tmpDataSend[66] := WORD_TO_BYTE(SHR(下卷扬伺服电流, 8));
tmpDataSend[67] := WORD_TO_BYTE(下卷扬伺服电流 AND 16#FF);
tmpDataSend[68] := WORD_TO_BYTE(SHR(下卷扬伺服速度, 8));
tmpDataSend[69] := WORD_TO_BYTE(下卷扬伺服速度 AND 16#FF);
tmpDataSend[70] := WORD_TO_BYTE(SHR(下卷扬伺服位置, 8));
tmpDataSend[71] := WORD_TO_BYTE(下卷扬伺服位置 AND 16#FF);
tmpDataSend[72] := WORD_TO_BYTE(SHR(下卷扬伺服温度, 8));
tmpDataSend[73] := WORD_TO_BYTE(下卷扬伺服温度 AND 16#FF);
tmpDataSend[74] := WORD_TO_BYTE(SHR(下卷扬伺服报错码, 8));
tmpDataSend[75] := WORD_TO_BYTE(下卷扬伺服报错码 AND 16#FF);
tmpDataSend[76] := 16#01;	//0-离线 1-在线

tmpDataSend[77] := WORD_TO_BYTE(SHR(滚刷伺服电流, 8));
tmpDataSend[78] := WORD_TO_BYTE(滚刷伺服电流 AND 16#FF);
tmpDataSend[79] := WORD_TO_BYTE(SHR(滚刷伺服速度, 8));
tmpDataSend[80] := WORD_TO_BYTE(滚刷伺服速度 AND 16#FF);
tmpDataSend[81] := WORD_TO_BYTE(SHR(滚刷伺服温度, 8));
tmpDataSend[82] := WORD_TO_BYTE(滚刷伺服温度 AND 16#FF);
tmpDataSend[83] := WORD_TO_BYTE(SHR(滚刷伺服报错码, 8));
tmpDataSend[84] := WORD_TO_BYTE(滚刷伺服报错码 AND 16#FF);
tmpDataSend[85] := 16#01;	//0-离线 1-在线

tmpDataSend[86] := 16#00;	//风机1启动状态 0-停止 1-启动
tmpDataSend[87] := 16#00;	//风机2启动状态 0-停止 1-启动

tmpDataSend[88] := WORD_TO_BYTE(SHR(左前测距超声波数据, 8));
tmpDataSend[89] := WORD_TO_BYTE(左前测距超声波数据 AND 16#FF);
tmpDataSend[90] := WORD_TO_BYTE(SHR(右前测距超声波数据, 8));
tmpDataSend[97] := WORD_TO_BYTE(右前测距超声波数据 AND 16#FF);
tmpDataSend[92] := WORD_TO_BYTE(SHR(左后测距超声波数据, 8));
tmpDataSend[93] := WORD_TO_BYTE(左后测距超声波数据 AND 16#FF);
tmpDataSend[94] := WORD_TO_BYTE(SHR(右后测距超声波数据, 8));
tmpDataSend[95] := WORD_TO_BYTE(右后测距超声波数据 AND 16#FF);

tmpDataSend[96] := WORD_TO_BYTE(SHR(左前边沿超声波数据, 8));
tmpDataSend[97] := WORD_TO_BYTE(左前边沿超声波数据 AND 16#FF);
tmpDataSend[98] := WORD_TO_BYTE(SHR(右前边沿超声波数据, 8));
tmpDataSend[99] := WORD_TO_BYTE(右前边沿超声波数据 AND 16#FF);
tmpDataSend[100] := WORD_TO_BYTE(SHR(左后边沿超声波数据, 8));
tmpDataSend[101] := WORD_TO_BYTE(左后边沿超声波数据 AND 16#FF);
tmpDataSend[102] := WORD_TO_BYTE(SHR(右后边沿超声波数据, 8));
tmpDataSend[103] := WORD_TO_BYTE(右后边沿超声波数据 AND 16#FF);

tmpDataSend[104] := WORD_TO_BYTE(SHR(机械臂空间X, 8));
tmpDataSend[105] := WORD_TO_BYTE(机械臂空间X AND 16#FF);
tmpDataSend[106] := WORD_TO_BYTE(SHR(机械臂空间Y, 8));
tmpDataSend[107] := WORD_TO_BYTE(机械臂空间Y AND 16#FF);
tmpDataSend[108] := WORD_TO_BYTE(SHR(机械臂空间Z, 8));
tmpDataSend[109] := WORD_TO_BYTE(机械臂空间Z AND 16#FF);
tmpDataSend[110] := WORD_TO_BYTE(SHR(机械臂空间B, 8));
tmpDataSend[111] := WORD_TO_BYTE(机械臂空间B AND 16#FF);
tmpDataSend[112] := WORD_TO_BYTE(SHR(底盘俯仰角, 8));
tmpDataSend[113] := WORD_TO_BYTE(底盘俯仰角 AND 16#FF);
tmpDataSend[114] := WORD_TO_BYTE(SHR(底盘横滚角, 8));
tmpDataSend[115] := WORD_TO_BYTE(底盘横滚角 AND 16#FF);

tmpDataSend[116] := WORD_TO_BYTE(机械臂运行状态); //0-上使能，1-掉使能，2-运行中，3-报错
tmpDataSend[117] := WORD_TO_BYTE(机械臂报错码);

上传信息处理_1(定时时间:=T#0MS, 数据域长度:=118, pInputData:=ADR(tmpDataSend[0]), 应答:=16#00, 序列号:=上传序列号, 主功能码:=16#02, 次功能码:=16#06);
END_METHOD

END_PROGRAM

// Device/Application/函数/运动控制/清扫作业流程
FUNCTION_BLOCK 清扫作业流程
VAR_IN_OUT
	作业状态		: INT;	//0-系统初始化, 10-清扫待命状态, 20-清扫准备状态, 30-清扫暂停状态, 40-行走复位状态, 50-急停状态, 60-进入现场操作模式, 70-退出现场操作模式
END_VAR
VAR_INPUT
	离地高度		: LREAL;
	光伏板角度		: LREAL;
	离车间距		: LREAL;
	清扫方向		: LREAL; //0-左侧, 1-右侧	
END_VAR
VAR_OUTPUT
	返回功能码		: BYTE;
	返回状态		: BYTE;		//0x00-运行中, 0x05-完成, 0x0A-异常
END_VAR
VAR
	机械臂清扫准备状态完成		: BOOL := FALSE;
END_VAR

CASE 作业状态 OF
	0 : //系统初始化
		滚刷伺服参数.运行模式 := 0;
		启动回零自动运行:=FALSE;
		启动对中机构自动运行:=FALSE;
		启动上下扬自动运行:=FALSE;
		作业状态 := 5;
	5:
	    启动回零自动运行:=TRUE;
		作业状态 := 6;
	6:
	    IF 回零工作完成 THEN
			返回功能码 := 16#01;
			返回状态 := 16#05;
	    END_IF
	10 : //清扫待命状态
		启动回零自动运行:=TRUE;
		IF 回零工作完成 THEN
            作业状态 := 11;
	    END_IF
	11 :
		机械臂运行参数.倍率 := 70.0;
		机械臂运行参数.规划模式 := 4;
		机械臂运行参数.是否关节运动 := TRUE;
		IF 清扫方向=1 THEN
			机械臂运行参数.运行点位[0] := 90.0;
		ELSE
			机械臂运行参数.运行点位[0] := -90.0;
		END_IF
		机械臂运行参数.运行点位[1] := -90.0; 机械臂运行参数.运行点位[2] := 180.0;
		机械臂运行参数.运行点位[3] := 50.0; 机械臂运行参数.运行点位[4] := 0.0; 机械臂运行参数.运行点位[5] := 0.0;
		IF sMotionOutputs.iRobStatus = 1 THEN
			机械臂运行启动 := TRUE;
		END_IF
		IF sMotionOutputs.iRobStatus = 3 THEN //运动完成
			返回功能码 := 16#02;
			返回状态 := 16#05;
		END_IF
	20 : //清扫准备状态
		机械臂运行参数.规划模式 := 4;
		机械臂运行参数.是否关节运动 := FALSE;
		IF 清扫方向=1 THEN
			机械臂运行参数.运行点位[1] := 2220.0;
		ELSE
			机械臂运行参数.运行点位[1] := -2220.0;
		END_IF
		机械臂运行参数.运行点位[0] := 0.0; 机械臂运行参数.运行点位[2] := 2000.0;
		机械臂运行参数.运行点位[3] := 40.0; 机械臂运行参数.运行点位[4] := 0.0; 机械臂运行参数.运行点位[5] := 0.0;
		滚刷伺服参数.运行模式 := 0;
		IF sMotionOutputs.iRobStatus = 1 THEN //机械臂运行至光伏板上方
			机械臂运行启动 := TRUE;
		END_IF
		IF sMotionOutputs.iRobStatus = 3 THEN //运动完成
			启动对中机构自动运行:=TRUE;
			作业状态 := 27;
		END_IF
	27:
	    IF 对中工作完成 THEN
			启动上下扬自动运行:=TRUE;
	    	作业状态 := 28;
	    END_IF
	28:
	    IF 上下卷扬工作完成 THEN
	    	作业状态 := 29;
	    END_IF
	29:	//清扫准备状态结束
// 	    滚刷伺服参数.运行方向:=TRUE;
		滚刷伺服参数.运行模式 := 1;
		IF 清扫方向=1 THEN
			滚刷伺服参数.运行方向:=FALSE;
		ELSE
			滚刷伺服参数.运行方向:=TRUE;
		END_IF
		返回功能码 := 16#03;
		返回状态 := 16#05;
	30 : //清扫暂停状态
		滚刷伺服参数.运行模式 := 0;
		//伸缩轴伺服参数.运行模式:=0;
		启动对中机构自动运行:=FALSE;
		启动上下扬自动运行:=FALSE;
		启动回零自动运行:=TRUE;
		IF 回零工作完成 THEN
			返回功能码 := 16#04;
			返回状态 := 16#05;
	    END_IF
	40 : //行走复位状态
		启动回零自动运行:=TRUE;
		IF 回零工作完成 THEN
            作业状态 := 41;
	    END_IF
	41 :
		机械臂运行参数.规划模式 := 4;
		机械臂运行参数.是否关节运动 := TRUE;
		机械臂运行参数.运行点位[0] := 0.0; 机械臂运行参数.运行点位[1] := -90.0; 机械臂运行参数.运行点位[2] := 180.0;
		机械臂运行参数.运行点位[3] := 45.0; 机械臂运行参数.运行点位[4] := 0.0; 机械臂运行参数.运行点位[5] := 0.0;
		IF sMotionOutputs.iRobStatus = 1 THEN
			机械臂运行启动 := TRUE;
		END_IF
		IF sMotionOutputs.iRobStatus = 3 THEN //运动完成
			返回功能码 := 16#05;
			返回状态 := 16#05;
		END_IF
	50 : //急停状态
		左上轮伺服参数.运行模式 := 0; 左下轮伺服参数.运行模式 := 0;
		右上轮伺服参数.运行模式 := 0; 右下轮伺服参数.运行模式 := 0;
	
	100: //无操作
// 		启动对中机构自动运行:=FALSE;
// 		启动上下扬自动运行:=FALSE;
		返回功能码 := 16#00;
		返回状态 := 16#00;
	200: //运行异常
		返回状态 := 16#0A;
ELSE
   滚刷伺服参数.运行模式 :=0;
   启动对中机构自动运行:=FALSE;
   启动上下扬自动运行:=FALSE;
END_CASE

END_FUNCTION_BLOCK

// Device/Application/底盘算法处理
PROGRAM 底盘算法处理
VAR
	iCounter			: INT := 0;
	底盘使能				: BOOL := FALSE;
	底盘联动				: BOOL := TRUE;
	
	底盘平衡处理			: 底盘平衡算法;
	
	左上气缸伺服控制    	: 伺服控制;
	左下气缸伺服控制    	: 伺服控制;
	右上气缸伺服控制    	: 伺服控制;
	右下气缸伺服控制    	: 伺服控制;
	
	左上轮伺服控制    	: 伺服控制;
	左下轮伺服控制    	: 伺服控制;
	右上轮伺服控制    	: 伺服控制;
	右下轮伺服控制    	: 伺服控制;  
END_VAR

底盘陀螺仪.X := DINT_TO_REAL(DWORD_TO_DINT( SHL(WORD_TO_DWORD(底盘陀螺仪.orign_arry[1]), 16) OR WORD_TO_DWORD(底盘陀螺仪.orign_arry[0]) )) / 1000;
底盘陀螺仪.Y := DINT_TO_REAL(DWORD_TO_DINT( SHL(WORD_TO_DWORD(底盘陀螺仪.orign_arry[3]), 16) OR WORD_TO_DWORD(底盘陀螺仪.orign_arry[2]) )) / 1000;
底盘陀螺仪.Z := DINT_TO_REAL(DWORD_TO_DINT( SHL(WORD_TO_DWORD(底盘陀螺仪.orign_arry[5]), 16) OR WORD_TO_DWORD(底盘陀螺仪.orign_arry[4]) )) / 1000;

底盘陀螺仪.角速度X := WORD_TO_REAL(底盘陀螺仪.orign_arry_speed[1]) / 32768 * 2000;
底盘陀螺仪.角速度Y := WORD_TO_REAL(底盘陀螺仪.orign_arry_speed[2]) / 32768 * 2000;
底盘陀螺仪.角速度Z := WORD_TO_REAL(底盘陀螺仪.orign_arry_speed[3]) / 32768 * 2000;

IF 底盘算法运行 THEN
	底盘平衡处理(
		陀螺仪roll:= 底盘陀螺仪.X, 
		陀螺仪pitch:= 底盘陀螺仪.Y, 
		陀螺仪roll速度:= 底盘陀螺仪.角速度X, 
		陀螺仪pitch速度:= 底盘陀螺仪.角速度Y, 
		前左轮实际长度:= 底盘控制.平均数据1,//左上气缸伺服参数.反馈位置, 
		后左轮实际长度:= 底盘控制.平均数据2,//左下气缸伺服参数.反馈位置, 	
		前右轮实际长度:= 底盘控制.平均数据3,//右上气缸伺服参数.反馈位置, 
		后右轮实际长度:= 底盘控制.平均数据4,//右下气缸伺服参数.反馈位置, 
		前左轮行驶速度:= 左上轮伺服参数.指令速度, 
		后左轮行驶速度:= 左下轮伺服参数.指令速度, 	
		前右轮行驶速度:= 右上轮伺服参数.指令速度, 
		后右轮行驶速度:= 右下轮伺服参数.指令速度, 	
		前左轮力:= 左上气缸伺服参数.反馈力矩, 
		后左轮力:= 左下气缸伺服参数.反馈力矩, 
		前右轮力:= 右上气缸伺服参数.反馈力矩, 
		后右轮力:= 右下气缸伺服参数.反馈力矩, 	
		前左轮输出=> 左上气缸伺服参数.运行位置, 
		后左轮输出=> 左下气缸伺服参数.运行位置, 
		前右轮输出=> 右上气缸伺服参数.运行位置, 
		后右轮输出=> 右下气缸伺服参数.运行位置,
		前左轮速度=> , 
		后左轮速度=> , 
		前右轮速度=> , 
		后右轮速度=> , );
END_IF

END_PROGRAM

// Device/Application/报警处理
PROGRAM 报警处理
VAR
	
END_VAR

DCH报警代码1:=报警代码1+报警代码2*255;
DCH报警代码2:=报警代码3+报警代码4*255;

// IF DCH遥控控制.DCH无线状态=FALSE THEN
// 	IF 报警代码2.1 THEN
// 		控制方式 := 1;	//自动模式
//     ELSE
// 	    控制方式 := 0;	//手动模式
// 	END_IF;
// END_IF

IF 伸缩轴.nAxisState=0 OR 上卷扬.nAxisState=0 OR 下卷扬.nAxisState=0 OR 滚刷.nAxisState=0
	OR 机械臂1轴.nAxisState=0 OR 机械臂2轴.nAxisState=0 OR 机械臂3轴.nAxisState=0 OR 机械臂4轴.nAxisState=0
	OR 右上气缸.nAxisState=0 OR 右下气缸.nAxisState=0 OR 左上气缸.nAxisState=0 OR 左下气缸.nAxisState=0
	OR 右上轮.nAxisState=0 OR 右下轮.nAxisState=0 OR 左上轮.nAxisState=0 OR 左下轮.nAxisState=0
	OR 伸缩轴.nAxisState=2 OR 上卷扬.nAxisState=2 OR 下卷扬.nAxisState=2 OR 滚刷.nAxisState=2
	OR 机械臂1轴.nAxisState=2 OR 机械臂2轴.nAxisState=2 OR 机械臂3轴.nAxisState=2 OR 机械臂4轴.nAxisState=2
	OR 右上气缸.nAxisState=2 OR 右下气缸.nAxisState=2 OR 左上气缸.nAxisState=2 OR 左下气缸.nAxisState=2
	OR 右上轮.nAxisState=2 OR 右下轮.nAxisState=2 OR 左上轮.nAxisState=2 OR 左下轮.nAxisState=2 THEN
	绿灯:=FALSE;
	黄灯:=TRUE;
	蜂鸣器:=FALSE;
ELSIF 伸缩轴.nAxisState<>0 AND 伸缩轴.nAxisState<>1 AND 伸缩轴.nAxisState<>2 
      AND 上卷扬.nAxisState<>0 AND 上卷扬.nAxisState<>1 AND 上卷扬.nAxisState<>2
	  AND 下卷扬.nAxisState<>0 AND 下卷扬.nAxisState<>1 AND 下卷扬.nAxisState<>2
	  AND 滚刷.nAxisState<>0 AND 滚刷.nAxisState<>1 AND 滚刷.nAxisState<>2
	  AND 机械臂1轴.nAxisState<>0 AND 机械臂1轴.nAxisState<>1 AND 机械臂1轴.nAxisState<>2
	  AND 机械臂2轴.nAxisState<>0 AND 机械臂2轴.nAxisState<>1 AND 机械臂2轴.nAxisState<>2
	  AND 机械臂3轴.nAxisState<>0 AND 机械臂3轴.nAxisState<>1 AND 机械臂3轴.nAxisState<>2
	  AND 机械臂4轴.nAxisState<>0 AND 机械臂4轴.nAxisState<>1 AND 机械臂4轴.nAxisState<>2
	  AND 右上气缸.nAxisState<>0 AND 右上气缸.nAxisState<>1 AND 右上气缸.nAxisState<>2
	  AND 右下气缸.nAxisState<>0 AND 右下气缸.nAxisState<>1 AND 右下气缸.nAxisState<>2
	  AND 左上气缸.nAxisState<>0 AND 左上气缸.nAxisState<>1 AND 左上气缸.nAxisState<>2
	  AND 左下气缸.nAxisState<>0 AND 左下气缸.nAxisState<>1 AND 左下气缸.nAxisState<>2
	  AND 右上轮.nAxisState<>0 AND 右上轮.nAxisState<>1 AND 右上轮.nAxisState<>2
	  AND 右下轮.nAxisState<>0 AND 右下轮.nAxisState<>1 AND 右下轮.nAxisState<>2
	  AND 左上轮.nAxisState<>0 AND 左上轮.nAxisState<>1 AND 左上轮.nAxisState<>2
	  AND 左下轮.nAxisState<>0 AND 左下轮.nAxisState<>1 AND 左下轮.nAxisState<>2 THEN
	  绿灯:=TRUE;
	  黄灯:=FALSE;
	  蜂鸣器:=FALSE;
// ELSE
END_IF


IF 伸缩轴.nAxisState=1 OR 上卷扬.nAxisState=1 OR 下卷扬.nAxisState=1 OR 滚刷.nAxisState=1
	OR 机械臂1轴.nAxisState=1 OR 机械臂2轴.nAxisState=1 OR 机械臂3轴.nAxisState=1 OR 机械臂4轴.nAxisState=1
	OR 右上气缸.nAxisState=1 OR 右下气缸.nAxisState=1 OR 左上气缸.nAxisState=1 OR 左下气缸.nAxisState=1
	OR 右上轮.nAxisState=1 OR 右下轮.nAxisState=1 OR 左上轮.nAxisState=1 OR 左下轮.nAxisState=1 THEN
	绿灯:=FALSE;
	黄灯:=FALSE;
	蜂鸣器:=TRUE;
	伸缩轴伺服参数.停止控制:=TRUE;    
	伸缩轴伺服参数.运行模式:=0;
    上卷扬伺服参数.停止控制:=TRUE;   
	上卷扬伺服参数.运行模式:=0;
    下卷扬伺服参数.停止控制:=TRUE; 
	下卷扬伺服参数.运行模式:=0;
    滚刷伺服参数.停止控制:=TRUE;  
	滚刷伺服参数.运行模式:=0;
    
    左上气缸伺服参数.停止控制:=TRUE; 
	左上气缸伺服参数.运行模式:=0;
    左下气缸伺服参数.停止控制:=TRUE; 
	左下气缸伺服参数.运行模式:=0;
    右上气缸伺服参数.停止控制:=TRUE;
	右上气缸伺服参数.运行模式:=0;
    右下气缸伺服参数.停止控制:=TRUE;    
	右下气缸伺服参数.运行模式:=0;
    
    左上轮伺服参数.停止控制:=TRUE;    
	左上轮伺服参数.运行模式:=0;
    左下轮伺服参数.停止控制:=TRUE;  
	左下轮伺服参数.运行模式:=0;
    右上轮伺服参数.停止控制:=TRUE;  
	右上轮伺服参数.运行模式:=0;
    右下轮伺服参数.停止控制:=TRUE;
	右下轮伺服参数.运行模式:=0;
	
	机械臂运行参数.规划模式:=5;
	机械臂运行启动:=1;
	轴报警:=TRUE;
ELSE
    轴报警:=FALSE;
END_IF
IF 报警复位 THEN
	IF 伸缩轴.nAxisState=1 THEN
		伸缩轴伺服参数.轴复位:=TRUE;
		//IF 伸缩轴伺服参数.复位状态.DONE AND 伸缩轴.nAxisState=1 THEN
		    伸缩轴伺服参数.轴初始化:=TRUE;
		//END_IF
	ELSE
	    伸缩轴伺服参数.轴复位:=FALSE;
		伸缩轴伺服参数.轴初始化:=FALSE;	
	END_IF
	IF 上卷扬.nAxisState=1 THEN
		上卷扬伺服参数.轴复位:=TRUE;
		//IF 上卷扬伺服参数.复位状态.DONE AND 上卷扬.nAxisState=1 THEN
		    上卷扬伺服参数.轴初始化:=TRUE;
		//END_IF
	ELSE
	    上卷扬伺服参数.轴复位:=FALSE;
		上卷扬伺服参数.轴初始化:=FALSE;	
	END_IF
	IF 下卷扬.nAxisState=1 THEN
		下卷扬伺服参数.轴复位:=TRUE;
		//IF 下卷扬伺服参数.复位状态.DONE AND 下卷扬.nAxisState=1 THEN
		    下卷扬伺服参数.轴初始化:=TRUE;
		//END_IF
	ELSE
	    下卷扬伺服参数.轴复位:=FALSE;
		下卷扬伺服参数.轴初始化:=FALSE;	
	END_IF
	IF 滚刷.nAxisState=1 THEN
		滚刷伺服参数.轴复位:=TRUE;
		//IF 滚刷伺服参数.复位状态.DONE AND 滚刷.nAxisState=1 THEN
		    滚刷伺服参数.轴初始化:=TRUE;
		//END_IF
	ELSE
	    滚刷伺服参数.轴复位:=FALSE;
		滚刷伺服参数.轴初始化:=FALSE;	
	END_IF
	IF 右上气缸.nAxisState=1 THEN
		右上气缸伺服参数.轴复位:=TRUE;
		//IF 右上气缸伺服参数.复位状态.DONE AND 右上气缸.nAxisState=1 THEN
		    右上气缸伺服参数.轴初始化:=TRUE;
		//END_IF
	ELSE
	    右上气缸伺服参数.轴复位:=FALSE;
		右上气缸伺服参数.轴初始化:=FALSE;	
	END_IF
	IF 右下气缸.nAxisState=1 THEN
		右上气缸伺服参数.轴复位:=TRUE;
		//IF 右下气缸伺服参数.复位状态.DONE AND 右下气缸.nAxisState=1 THEN
		    右下气缸伺服参数.轴初始化:=TRUE;
		//END_IF
	ELSE
	    右下气缸伺服参数.轴复位:=FALSE;
		右下气缸伺服参数.轴初始化:=FALSE;	
	END_IF
	IF 左上气缸.nAxisState=1 THEN
		右上气缸伺服参数.轴复位:=TRUE;
		//IF 左上气缸伺服参数.复位状态.DONE AND 左上气缸.nAxisState=1 THEN
		    左上气缸伺服参数.轴初始化:=TRUE;
		//END_IF
	ELSE
	    左上气缸伺服参数.轴复位:=FALSE;
		左上气缸伺服参数.轴初始化:=FALSE;	
	END_IF
	IF 左下气缸.nAxisState=1 THEN
		右上气缸伺服参数.轴复位:=TRUE;
		//IF 左下气缸伺服参数.复位状态.DONE AND 左下气缸.nAxisState=1 THEN
		    左下气缸伺服参数.轴初始化:=TRUE;
		//END_IF
	ELSE
	    左下气缸伺服参数.轴复位:=FALSE;
		左下气缸伺服参数.轴初始化:=FALSE;	
	END_IF
	IF 右上轮.nAxisState=1 THEN
		右上轮伺服参数.轴复位:=TRUE;
		//IF 右上轮伺服参数.复位状态.DONE AND 右上轮.nAxisState=1 THEN
		    右上轮伺服参数.轴初始化:=TRUE;
		//END_IF
	ELSE
	    右上轮伺服参数.轴复位:=FALSE;
		右上轮伺服参数.轴初始化:=FALSE;	
	END_IF
	IF 右下轮.nAxisState=1 THEN
		右下轮伺服参数.轴复位:=TRUE;
		//IF 右下轮伺服参数.复位状态.DONE AND 右下轮.nAxisState=1 THEN
		    右下轮伺服参数.轴初始化:=TRUE;
		//END_IF
	ELSE
	    右下轮伺服参数.轴复位:=FALSE;
		右下轮伺服参数.轴初始化:=FALSE;	
	END_IF
	IF 左上轮.nAxisState=1 THEN
		左上轮伺服参数.轴复位:=TRUE;
		//IF 左上轮伺服参数.复位状态.DONE AND 左上轮.nAxisState=1 THEN
		    左上轮伺服参数.轴初始化:=TRUE;
		//END_IF
	ELSE
	    左上轮伺服参数.轴复位:=FALSE;
		左上轮伺服参数.轴初始化:=FALSE;	
	END_IF
	IF 左下轮.nAxisState=1 THEN
		左下轮伺服参数.轴复位:=TRUE;
		//IF 左下轮伺服参数.复位状态.DONE AND 左下轮.nAxisState=1 THEN
		    左下轮伺服参数.轴初始化:=TRUE;
		//END_IF
	ELSE
	    左下轮伺服参数.轴复位:=FALSE;
		左下轮伺服参数.轴初始化:=FALSE;	
	END_IF
	IF 机械臂1轴.nAxisState=1 OR 机械臂2轴.nAxisState=1 OR 机械臂3轴.nAxisState=1 OR 机械臂4轴.nAxisState=1 THEN
		;//机械臂控制.报错复位:=TRUE;
	END_IF
ELSE
    伸缩轴伺服参数.轴复位:=FALSE;
	伸缩轴伺服参数.轴初始化:=FALSE;
	上卷扬伺服参数.轴复位:=FALSE;
	上卷扬伺服参数.轴初始化:=FALSE;	
	下卷扬伺服参数.轴复位:=FALSE;
	下卷扬伺服参数.轴初始化:=FALSE;
	滚刷伺服参数.轴复位:=FALSE;
	滚刷伺服参数.轴初始化:=FALSE;
	右上气缸伺服参数.轴复位:=FALSE;
	右上气缸伺服参数.轴初始化:=FALSE;	
	右下气缸伺服参数.轴复位:=FALSE;
	右下气缸伺服参数.轴初始化:=FALSE;
	左上轮伺服参数.轴复位:=FALSE;
	左上轮伺服参数.轴初始化:=FALSE;	
	左下轮伺服参数.轴复位:=FALSE;
	左下轮伺服参数.轴初始化:=FALSE;	
END_IF
(*
//限位
/////////////////////////////////////////////////////
//伸缩轴
IF (伸缩轴.fActPosition>伸缩架上限位 OR 伸缩轴.fActPosition<伸缩架下限位) AND 控制方式=1 THEN
	伸缩轴伺服参数.停止控制:=TRUE;
	伸缩轴伺服参数.运行模式:=0;
	伸缩架限位报警:=TRUE;
ELSIF (伸缩轴.fActPosition>伸缩架上限位 OR 伸缩轴.fActPosition<伸缩架下限位) AND 控制方式=0 THEN
    伸缩架限位报警:=TRUE;
ELSE
    伸缩架限位报警:=FALSE;
END_IF
//上卷扬
IF (上卷扬.fActPosition>上卷扬上限位 OR 上卷扬.fActPosition<上卷扬下限位) AND 控制方式=1 THEN
	上卷扬伺服参数.停止控制:=TRUE;
	上卷扬伺服参数.运行模式:=0;
	上卷扬限位报警:=TRUE;
ELSIF (上卷扬.fActPosition>上卷扬上限位 OR 上卷扬.fActPosition<上卷扬下限位) AND 控制方式=0 THEN
    上卷扬限位报警:=TRUE;
ELSE
    上卷扬限位报警:=FALSE;
END_IF
//下卷扬
IF (下卷扬.fActPosition>伸缩架上限位 OR 下卷扬.fActPosition<下卷扬下限位) AND 控制方式=1 THEN
	下卷扬伺服参数.停止控制:=TRUE;
	下卷扬伺服参数.运行模式:=0;
	下卷扬限位报警:=TRUE;
ELSIF (下卷扬.fActPosition>下卷扬上限位 OR 下卷扬.fActPosition<下卷扬下限位) AND 控制方式=0 THEN
    下卷扬限位报警:=TRUE;
ELSE
    下卷扬限位报警:=FALSE;
END_IF
//左上气缸
IF (左上气缸.fActPosition>左上气缸上限位 OR 左上气缸.fActPosition<左上气缸下限位) AND 控制方式=1 THEN
	左上气缸伺服参数.停止控制:=TRUE;
	左上气缸伺服参数.运行模式:=0;
	左上气缸限位报警:=TRUE;
ELSIF (左上气缸.fActPosition>左上气缸上限位 OR 左上气缸.fActPosition<左上气缸下限位) AND 控制方式=0 THEN
    左上气缸限位报警:=TRUE;
ELSE
    左上气缸限位报警:=FALSE;
END_IF
//左下气缸
IF (左下气缸.fActPosition>左下气缸上限位 OR 左下气缸.fActPosition<左下气缸下限位) AND 控制方式=1 THEN
	左下气缸伺服参数.停止控制:=TRUE;
	左下气缸伺服参数.运行模式:=0;
	左下气缸限位报警:=TRUE;
ELSIF (左下气缸.fActPosition>左下气缸上限位 OR 左下气缸.fActPosition<左下气缸下限位) AND 控制方式=0 THEN
    左下气缸限位报警:=TRUE;
ELSE
    左下气缸限位报警:=FALSE;
END_IF
//右上气缸
IF (右上气缸.fActPosition>右上气缸上限位 OR 右上气缸.fActPosition<右上气缸下限位) AND 控制方式=1 THEN
	右上气缸伺服参数.停止控制:=TRUE;
	右上气缸伺服参数.运行模式:=0;
	右上气缸限位报警:=TRUE;
ELSIF (右上气缸.fActPosition>右上气缸上限位 OR 右上气缸.fActPosition<右上气缸下限位) AND 控制方式=0 THEN
    右上气缸限位报警:=TRUE;
ELSE
    右上气缸限位报警:=FALSE;
END_IF
//右下气缸
IF (右下气缸.fActPosition>右下气缸上限位 OR 右下气缸.fActPosition<右下气缸下限位) AND 控制方式=1 THEN
	右下气缸伺服参数.停止控制:=TRUE;
	右下气缸伺服参数.运行模式:=0;
	右下气缸限位报警:=TRUE;
ELSIF (右下气缸.fActPosition>右下气缸上限位 OR 右下气缸.fActPosition<右下气缸下限位) AND 控制方式=0 THEN
    右下气缸限位报警:=TRUE;
ELSE
    右下气缸限位报警:=FALSE;
END_IF
*)

END_PROGRAM

// Device/Application/函数/运动控制/底盘控制运动
FUNCTION_BLOCK 底盘控制运动
VAR_INPUT
	启动底盘自动运行:BOOL;
	//pAxis      	: POINTER TO AXIS_REF_SM3;	//定义轴
	//实时运行位置:LREAL;
END_VAR
VAR_OUTPUT
END_VAR
VAR
	底盘控制自动流程:INT;
	位置记录1:LREAL;
	位置记录2:LREAL;
	delay1:INT;
	delay2:INT;
END_VAR
VAR_IN_OUT
	伺服参数    			: 伺服参数结构体;
END_VAR

IF 启动底盘自动运行 THEN
	CASE 底盘控制自动流程 OF
	0:
	   伺服参数.运行模式:=0;
	   delay1:=0;
	   delay2:=0;
	   底盘控制自动流程:=10;
	   
	   
	10:   
	  // delay2:=0;
	   位置记录1:=伺服参数.运行位置;
	   伺服参数.运行位置:=位置记录1;
	   伺服参数.运行模式:=2;
	   底盘控制自动流程:=20;
	20:  
	   //IF 伺服参数.运动到点完成 THEN
	 //  delay1:=delay1+1;
	  // IF delay1=5 THEN
	
	      位置记录2:=伺服参数.运行位置;
	   	  伺服参数.运行位置1:=位置记录2;
	      伺服参数.运行模式:=4;
	      底盘控制自动流程:=10;
	   //END_IF
	   //END_IF
	30:
	   //IF 伺服参数.运动到点完成1 THEN
	     // delay1:=0;
		//  delay2:=delay2+1;
        //  IF delay2=5 THEN
			
	      底盘控制自动流程:=10;
		//  END_IF
	   //END_IF
	 END_CASE
ELSE
     //伺服参数.运行模式:=0;
	 底盘控制自动流程:=0;
END_IF

END_FUNCTION_BLOCK

// Device/Application/函数/运动控制/底盘控制运动_1
FUNCTION_BLOCK 底盘控制运动_1
VAR_INPUT
	启动底盘自动运行:BOOL;
	//pAxis      	: POINTER TO AXIS_REF_SM3;	//定义轴
	//实时运行位置:LREAL;
END_VAR
VAR_OUTPUT
END_VAR
VAR
	底盘控制自动流程:INT;
	位置记录1:LREAL;
	位置记录2:LREAL;
	delay1:INT;
	delay2:INT;
END_VAR
VAR_IN_OUT
	伺服参数    			: 伺服参数结构体;
END_VAR

IF 启动底盘自动运行 THEN
	IF 伺服参数.运行速度=0 THEN
		底盘控制自动流程:=0;
	END_IF
	CASE 底盘控制自动流程 OF
	0:
	   伺服参数.运行模式:=0;
	   delay1:=0;
	   delay2:=0;
	   IF 伺服参数.运行速度<>0 THEN
	   	底盘控制自动流程:=10;
	   END_IF
	   
	   
	   
	10:   
	  // delay2:=0;
	   位置记录1:=伺服参数.运行速度;
	   伺服参数.运行控制速度:=ABS(位置记录1);
	   (*
	   IF 伺服参数.运行速度>0 THEN
	    伺服参数.运行控制方向:=1	;
	   ELSE
	    伺服参数.运行控制方向:=-1	;
	   END_IF
	   *)
	   伺服参数.运行模式:=6;
	   底盘控制自动流程:=20;
	20:  
	   //IF 伺服参数.运动到点完成 THEN
	 //  delay1:=delay1+1;
	  // IF delay1=5 THEN
	
	      位置记录2:=伺服参数.运行速度;
	   	  伺服参数.运行控制速度1:=ABS(位置记录2);
		  (*
		  IF 伺服参数.运行速度>0 THEN
			伺服参数.运行控制方向:=1	;
		   ELSE
			伺服参数.运行控制方向:=-1	;
		   END_IF
		   *)
	      伺服参数.运行模式:=7;
	      底盘控制自动流程:=10;
	   //END_IF
	   //END_IF
	30:
	   //IF 伺服参数.运动到点完成1 THEN
	     // delay1:=0;
		//  delay2:=delay2+1;
        //  IF delay2=5 THEN
			
	      底盘控制自动流程:=10;
		//  END_IF
	   //END_IF
	 END_CASE
ELSE
     //伺服参数.运行模式:=0;
	 底盘控制自动流程:=0;
END_IF

END_FUNCTION_BLOCK

// Device/Application/函数/运动控制/低通滤波模块
FUNCTION_BLOCK 低通滤波模块
VAR_INPUT
	输入数据		: LREAL;
	滤波系数		: LREAL := 0.3;
END_VAR
VAR_OUTPUT
	输出数据		: LREAL;
END_VAR
VAR
	上周期数据	: LREAL;
END_VAR

输出数据 := (1 - 滤波系数)*上周期数据 + 滤波系数*输入数据;
上周期数据 := 输出数据;

END_FUNCTION_BLOCK

// Device/Application/函数/运动控制/底盘控制运动_2
FUNCTION_BLOCK 底盘控制运动_2
VAR_INPUT
	启动底盘自动运行:BOOL;
	//pAxis      	: POINTER TO AXIS_REF_SM3;	//定义轴
	//实时运行位置:LREAL;
END_VAR
VAR_OUTPUT
END_VAR
VAR
	底盘控制自动流程:INT;
	位置记录1:LREAL;
	位置记录2:LREAL;
	delay1:INT;
	delay2:INT;
END_VAR
VAR_IN_OUT
	伺服参数    			: 伺服参数结构体;
END_VAR

IF 启动底盘自动运行 THEN
	CASE 底盘控制自动流程 OF
	0:
	   伺服参数.运行模式:=0;
	   delay1:=0;
	   delay2:=0;
	   底盘控制自动流程:=10;
	   
	10:   
	  // delay2:=0;
	   位置记录1:=伺服参数.运行力矩;
	   伺服参数.设定力矩:=位置记录1;
	   伺服参数.运行模式:=8;
	   底盘控制自动流程:=20;
	20:  
	   //IF 伺服参数.运动到点完成 THEN
	 //  delay1:=delay1+1;
	  // IF delay1=5 THEN
	
	      位置记录2:=伺服参数.运行力矩;
	   	  伺服参数.设定力矩1:=位置记录2;
	      伺服参数.运行模式:=9;
	      底盘控制自动流程:=10;
	   //END_IF
	   //END_IF
	30:
	   //IF 伺服参数.运动到点完成1 THEN
	     // delay1:=0;
		//  delay2:=delay2+1;
        //  IF delay2=5 THEN
			
	      底盘控制自动流程:=10;
		//  END_IF
	   //END_IF
	 END_CASE
ELSE
     //伺服参数.运行模式:=0;
	 底盘控制自动流程:=0;
END_IF

END_FUNCTION_BLOCK

// Device/Application/函数/运动控制/超声波实时检测调整
FUNCTION_BLOCK 超声波实时检测调整
VAR_INPUT
	超声波实时检测:BOOL;
	//pAxis      	: POINTER TO AXIS_REF_SM3;	//定义轴
	//实时运行位置:LREAL;
	运行位置		: LREAL;
END_VAR
VAR_OUTPUT
END_VAR
VAR
	超声波实时检测自动流程:INT;
	位置记录1:LREAL;
	位置记录2:LREAL;
	delay1:INT;
	delay2:INT;
END_VAR
VAR_IN_OUT
	伺服参数    			: 伺服参数结构体;
END_VAR

IF 超声波实时检测 THEN
	CASE 超声波实时检测自动流程 OF
	0:
	   伺服参数.运行模式:=0;
	   delay1:=0;
	   delay2:=0;
	   超声波实时检测自动流程:=10;
	   
	   
	10:   
	  // delay2:=0;
	   位置记录1:=运行位置;
	   伺服参数.运行位置:=位置记录1;
	   伺服参数.运行模式:=2;
	   超声波实时检测自动流程:=20;
	20:  
	   //IF 伺服参数.运动到点完成 THEN
	 //  delay1:=delay1+1;
	  // IF delay1=5 THEN
	
	      位置记录2:=运行位置;
	   	  伺服参数.运行位置1:=位置记录2;
	      伺服参数.运行模式:=4;
	      超声波实时检测自动流程:=10;
	   //END_IF
	   //END_IF
	30:
	   //IF 伺服参数.运动到点完成1 THEN
	     // delay1:=0;
		//  delay2:=delay2+1;
        //  IF delay2=5 THEN
			
	      超声波实时检测自动流程:=10;
		//  END_IF
	   //END_IF
	 END_CASE
ELSE
    // 伺服参数.运行模式:=0;
	 超声波实时检测自动流程:=0;
END_IF

END_FUNCTION_BLOCK
